FUNCTION_BLOCK ATV320 (* Composite Function Block Type *)
  (* Standard: 61499-2 *)
  (* Version 0.0, 06/08/2021, SESA371406, Schneider Electric, template *)
  PACKAGE SE.Nereda;
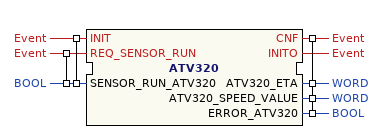
  EVENT_INPUT
    INIT WITH SENSOR_RUN_ATV320;
    REQ_SENSOR_RUN WITH SENSOR_RUN_ATV320;
  END_EVENT
  EVENT_OUTPUT
    CNF WITH ERROR_ATV320, ATV320_ETA, ATV320_SPEED_VALUE;
    INITO;
  END_EVENT
  VAR_INPUT
    SENSOR_RUN_ATV320 : BOOL;
  END_VAR
  VAR_OUTPUT
    ATV320_ETA : WORD;
    ATV320_SPEED_VALUE : WORD;
    ERROR_ATV320 : BOOL;
  END_VAR
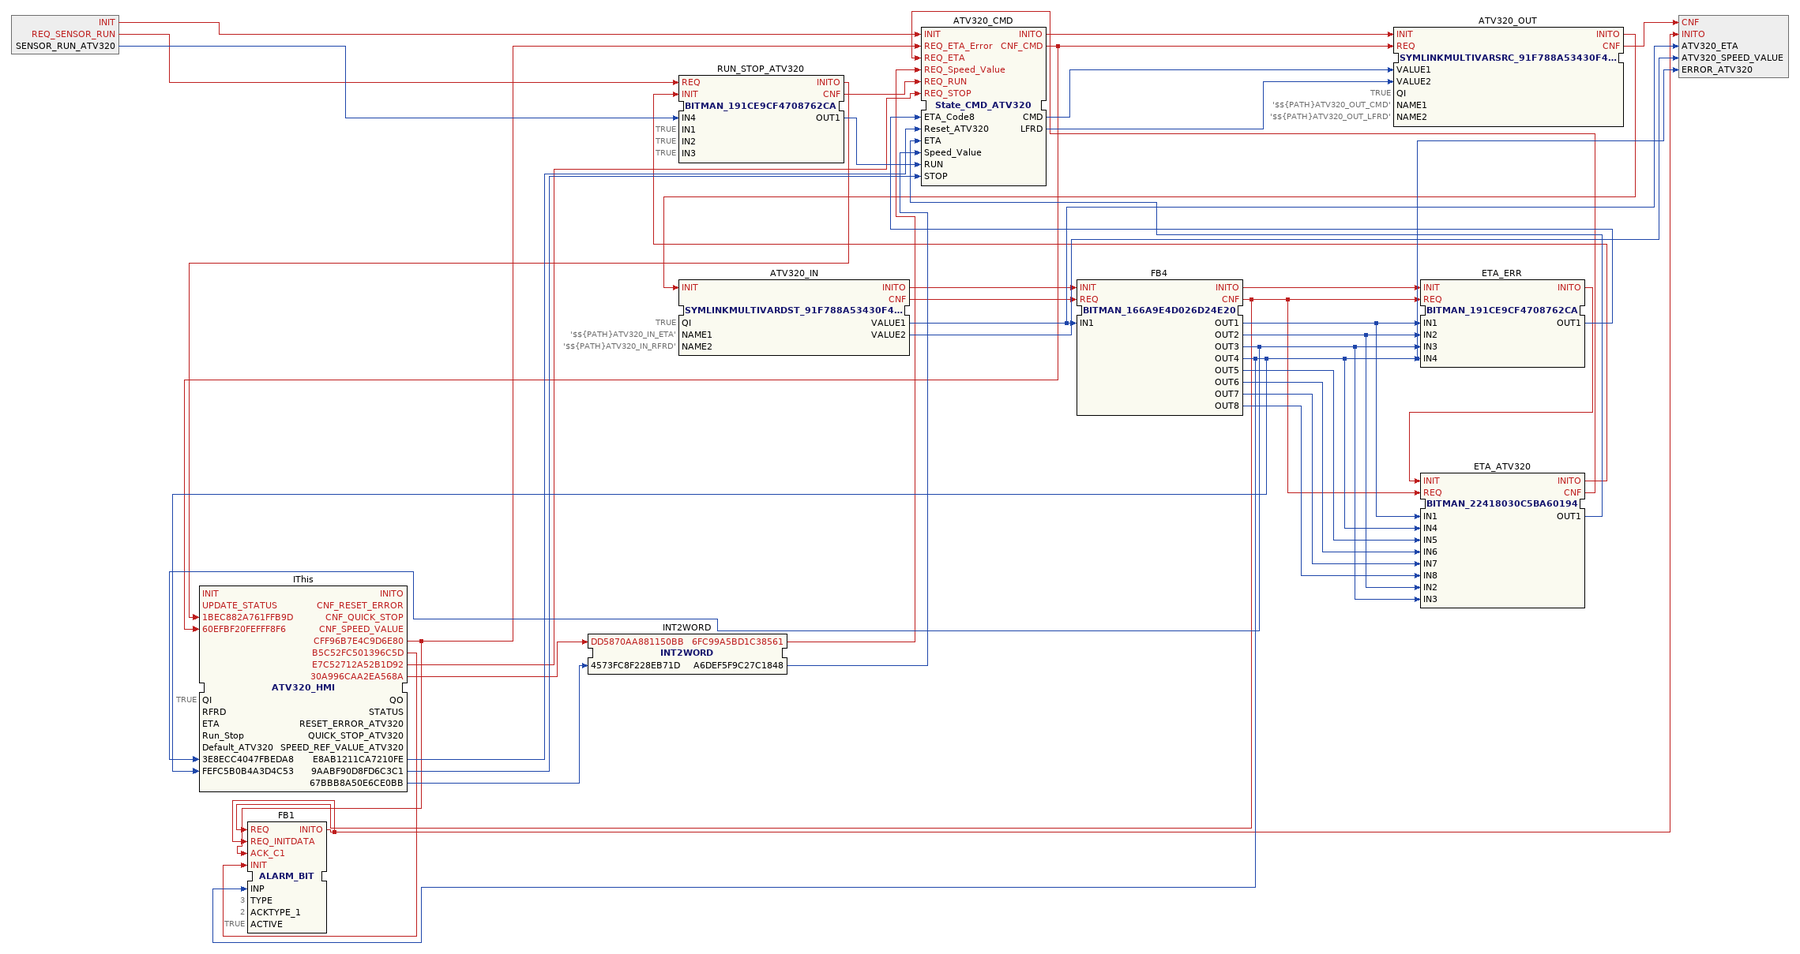
  FBS
    ATV320_IN : SYMLINKMULTIVARDST_91F788A53430F44E(QI := TRUE, NAME1 := '$${PATH}ATV320_IN_ETA' {SET_ATTRIBUTE(Configuration.Parameter.Style, Width=500)}, NAME2 := '$${PATH}ATV320_IN_RFRD' {SET_ATTRIBUTE(Configuration.Parameter.Style, Width=500)}); {SET_ATTRIBUTE(Configuration.GenericFBType.InterfaceParams, Runtime.System#I:=2;VALUE${I$}:WORD,WORD)}
    ATV320_OUT : SYMLINKMULTIVARSRC_91F788A53430F44E(QI := TRUE, NAME1 := '$${PATH}ATV320_OUT_CMD' {SET_ATTRIBUTE(Configuration.Parameter.Style, Width=500)}, NAME2 := '$${PATH}ATV320_OUT_LFRD' {SET_ATTRIBUTE(Configuration.Parameter.Style, Width=500)}); {SET_ATTRIBUTE(Configuration.GenericFBType.InterfaceParams, Runtime.System#I:=2;VALUE${I$}:WORD,WORD)}
    FB4 : BITMAN_166A9E4D026D24E20; {SET_ATTRIBUTE(Configuration.GenericFBType.InterfaceParams, Runtime.Standard#CNTIN:=1;CNTOUT:=8;IN${CNTIN$}:WORD;OUT${CNTOUT$}:BOOL,BOOL,BOOL,BOOL,BOOL,BOOL,BOOL,BOOL)}
    ETA_ERR : BITMAN_191CE9CF4708762CA; {SET_ATTRIBUTE(Configuration.GenericFBType.InterfaceParams, Runtime.Standard#CNTIN:=4;CNTOUT:=1;IN${CNTIN$}:BOOL,BOOL,BOOL,BOOL;OUT${CNTOUT$}:WORD)}
    ETA_ATV320 : BITMAN_22418030C5BA60194; {SET_ATTRIBUTE(Configuration.GenericFBType.InterfaceParams, Runtime.Standard#CNTIN:=8;CNTOUT:=1;IN${CNTIN$}:BOOL,BOOL,BOOL,BOOL,BOOL,BOOL,BOOL,BOOL;OUT${CNTOUT$}:WORD)}
    ATV320_CMD : State_CMD_ATV320;
    RUN_STOP_ATV320 : BITMAN_191CE9CF4708762CA(IN1 := TRUE, IN2 := TRUE, IN3 := TRUE); {SET_ATTRIBUTE(Configuration.GenericFBType.InterfaceParams, Runtime.Standard#CNTIN:=4;CNTOUT:=1;IN${CNTIN$}:BOOL,BOOL,BOOL,BOOL;OUT${CNTOUT$}:WORD)}
    IThis : ATV320_HMI(QI := TRUE);
    FB1 : ALARM_BIT(TYPE := 3, ACKTYPE_1 := 2, ACTIVE := TRUE);
    INT2WORD : INT2WORD;
  END_FBS
  EVENT_CONNECTIONS
    ATV320_OUT.INITO TO ATV320_IN.INIT;
    ATV320_IN.INITO TO FB4.INIT;
    ATV320_IN.CNF TO FB4.REQ;
    FB4.INITO TO ETA_ERR.INIT;
    FB4.CNF TO ETA_ERR.REQ;
    ETA_ERR.INITO TO ETA_ATV320.INIT;
    FB4.CNF TO ETA_ATV320.REQ;
    REQ_SENSOR_RUN TO RUN_STOP_ATV320.REQ;
    ATV320_OUT.CNF TO CNF;
    ETA_ATV320.INITO TO RUN_STOP_ATV320.INIT;
    FB4.CNF TO FB1.REQ;
    FB1.INITO TO FB1.REQ_INITDATA;
    RUN_STOP_ATV320.INITO TO IThis.1BEC882A761FFB9D;
    IThis.CFF96B7E4C9D6E80 TO FB1.ACK_C1;
    FB1.INITO TO INITO;
    IThis.B5C52FC501396C5D TO FB1.INIT;
    INIT TO ATV320_CMD.INIT;
    IThis.CFF96B7E4C9D6E80 TO ATV320_CMD.REQ_ETA_Error;
    ETA_ATV320.CNF TO ATV320_CMD.REQ_ETA;
    INT2WORD.6FC99A5BD1C38561 TO ATV320_CMD.REQ_Speed_Value;
    RUN_STOP_ATV320.CNF TO ATV320_CMD.REQ_RUN;
    IThis.E7C52712A52B1D92 TO ATV320_CMD.REQ_STOP;
    ATV320_CMD.INITO TO ATV320_OUT.INIT;
    ATV320_CMD.CNF_CMD TO ATV320_OUT.REQ;
    ATV320_CMD.CNF_CMD TO IThis.60EFBF20FEFFF8F6;
    IThis.30A996CAA2EA568A TO INT2WORD.DD5870AA881150BB;
  END_CONNECTIONS
  DATA_CONNECTIONS
    ATV320_IN.VALUE1 TO FB4.IN1;
    FB4.OUT1 TO ETA_ERR.IN1;
    FB4.OUT2 TO ETA_ERR.IN2;
    FB4.OUT3 TO ETA_ERR.IN3;
    FB4.OUT4 TO ETA_ERR.IN4;
    FB4.OUT1 TO ETA_ATV320.IN1;
    FB4.OUT4 TO ETA_ATV320.IN4;
    FB4.OUT5 TO ETA_ATV320.IN5;
    FB4.OUT6 TO ETA_ATV320.IN6;
    FB4.OUT7 TO ETA_ATV320.IN7;
    FB4.OUT8 TO ETA_ATV320.IN8;
    FB4.OUT2 TO ETA_ATV320.IN2;
    FB4.OUT3 TO ETA_ATV320.IN3;
    SENSOR_RUN_ATV320 TO RUN_STOP_ATV320.IN4;
    ATV320_IN.VALUE2 TO ATV320_SPEED_VALUE;
    ATV320_IN.VALUE1 TO ATV320_ETA;
    FB4.OUT4 TO ERROR_ATV320;
    FB4.OUT4 TO FB1.INP;
    FB4.OUT3 TO IThis.3E8ECC4047FBEDA8;
    FB4.OUT4 TO IThis.FEFC5B0B4A3D4C53;
    ETA_ERR.OUT1 TO ATV320_CMD.ETA_Code8;
    IThis.E8AB1211CA7210FE TO ATV320_CMD.Reset_ATV320;
    ETA_ATV320.OUT1 TO ATV320_CMD.ETA;
    INT2WORD.A6DEF5F9C27C1848 TO ATV320_CMD.Speed_Value;
    RUN_STOP_ATV320.OUT1 TO ATV320_CMD.RUN;
    IThis.9AABF90D8FD6C3C1 TO ATV320_CMD.STOP;
    ATV320_CMD.CMD TO ATV320_OUT.VALUE1;
    ATV320_CMD.LFRD TO ATV320_OUT.VALUE2;
    IThis.67BBB8A50E6CE0BB TO INT2WORD.4573FC8F228EB71D;
  END_CONNECTIONS
END_FUNCTION_BLOCK
